// TIA Portal V17 export
// export: Created 2024-01-16T10:06:36.9177276Z, ExportSetting None, DisplayName Totally Integrated Automation Portal, DisplayVersion V17 Update 4, DisplayName TIA Portal Openness, DisplayVersion V17 Update 4, DisplayName TIA Portal Version Control Interface, DisplayVersion V17, DisplayName STEP 7 Professional, DisplayVersion V17 Update 4, DisplayName STEP 7 Safety, DisplayVersion V17, DisplayName WinCC Advanced / Unified PC, DisplayVersion V17 Update 4
FUNCTION "FC_FDIn" : Void   // FC13, F_LAD
// stored: AutoNumber false
BEGIN

REGION Network 1: GAS INLET VALVE OPEN
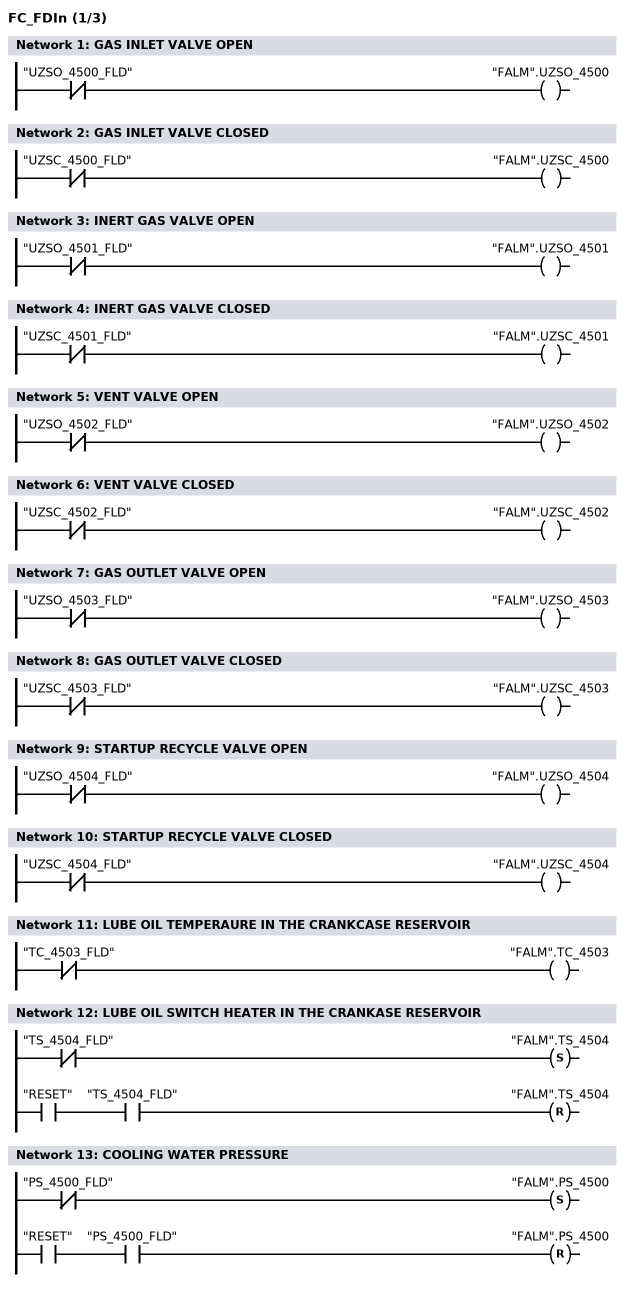
   RUNG wire#powerrail
      I_Contact( "UZSO_4500_FLD" )
      Coil( "FALM".UZSO_4500 )
   END_RUNG
   // the same network as SCL:
   "FALM".UZSO_4500 := NOT "UZSO_4500_FLD";
END_REGION

REGION Network 2: GAS INLET VALVE CLOSED
   RUNG wire#powerrail
      I_Contact( "UZSC_4500_FLD" )
      Coil( "FALM".UZSC_4500 )
   END_RUNG
   // the same network as SCL:
   "FALM".UZSC_4500 := NOT "UZSC_4500_FLD";
END_REGION

REGION Network 3: INERT GAS VALVE OPEN
   RUNG wire#powerrail
      I_Contact( "UZSO_4501_FLD" )
      Coil( "FALM".UZSO_4501 )
   END_RUNG
   // the same network as SCL:
   "FALM".UZSO_4501 := NOT "UZSO_4501_FLD";
END_REGION

REGION Network 4: INERT GAS VALVE CLOSED
   RUNG wire#powerrail
      I_Contact( "UZSC_4501_FLD" )
      Coil( "FALM".UZSC_4501 )
   END_RUNG
   // the same network as SCL:
   "FALM".UZSC_4501 := NOT "UZSC_4501_FLD";
END_REGION

REGION Network 5: VENT VALVE OPEN
   RUNG wire#powerrail
      I_Contact( "UZSO_4502_FLD" )
      Coil( "FALM".UZSO_4502 )
   END_RUNG
   // the same network as SCL:
   "FALM".UZSO_4502 := NOT "UZSO_4502_FLD";
END_REGION

REGION Network 6: VENT VALVE CLOSED
   RUNG wire#powerrail
      I_Contact( "UZSC_4502_FLD" )
      Coil( "FALM".UZSC_4502 )
   END_RUNG
   // the same network as SCL:
   "FALM".UZSC_4502 := NOT "UZSC_4502_FLD";
END_REGION

REGION Network 7: GAS OUTLET VALVE OPEN
   RUNG wire#powerrail
      I_Contact( "UZSO_4503_FLD" )
      Coil( "FALM".UZSO_4503 )
   END_RUNG
   // the same network as SCL:
   "FALM".UZSO_4503 := NOT "UZSO_4503_FLD";
END_REGION

REGION Network 8: GAS OUTLET VALVE CLOSED
   RUNG wire#powerrail
      I_Contact( "UZSC_4503_FLD" )
      Coil( "FALM".UZSC_4503 )
   END_RUNG
   // the same network as SCL:
   "FALM".UZSC_4503 := NOT "UZSC_4503_FLD";
END_REGION

REGION Network 9: STARTUP RECYCLE VALVE OPEN
   RUNG wire#powerrail
      I_Contact( "UZSO_4504_FLD" )
      Coil( "FALM".UZSO_4504 )
   END_RUNG
   // the same network as SCL:
   "FALM".UZSO_4504 := NOT "UZSO_4504_FLD";
END_REGION

REGION Network 10: STARTUP RECYCLE VALVE CLOSED
   RUNG wire#powerrail
      I_Contact( "UZSC_4504_FLD" )
      Coil( "FALM".UZSC_4504 )
   END_RUNG
   // the same network as SCL:
   "FALM".UZSC_4504 := NOT "UZSC_4504_FLD";
END_REGION

REGION Network 11: LUBE OIL TEMPERAURE IN THE CRANKCASE RESERVOIR
   RUNG wire#powerrail
      I_Contact( "TC_4503_FLD" )
      Coil( "FALM".TC_4503 )
   END_RUNG
   // the same network as SCL:
   "FALM".TC_4503 := NOT "TC_4503_FLD";
END_REGION

REGION Network 12: LUBE OIL SWITCH HEATER IN THE CRANKASE RESERVOIR
   RUNG wire#powerrail
      I_Contact( "TS_4504_FLD" )
      S_Coil( "FALM".TS_4504 )
   END_RUNG
   RUNG wire#powerrail
      Contact( "RESET" )
      Contact( "TS_4504_FLD" )
      R_Coil( "FALM".TS_4504 )
   END_RUNG
   // the same network as SCL:
   IF NOT "TS_4504_FLD" THEN "FALM".TS_4504 := TRUE; END_IF;
   IF "RESET" AND "TS_4504_FLD" THEN "FALM".TS_4504 := FALSE; END_IF;
END_REGION

REGION Network 13: COOLING WATER PRESSURE
   RUNG wire#powerrail
      I_Contact( "PS_4500_FLD" )
      S_Coil( "FALM".PS_4500 )
   END_RUNG
   RUNG wire#powerrail
      Contact( "RESET" )
      Contact( "PS_4500_FLD" )
      R_Coil( "FALM".PS_4500 )
   END_RUNG
   // the same network as SCL:
   IF NOT "PS_4500_FLD" THEN "FALM".PS_4500 := TRUE; END_IF;
   IF "RESET" AND "PS_4500_FLD" THEN "FALM".PS_4500 := FALSE; END_IF;
END_REGION

REGION Network 14: OUTLET GAS PRESSURE
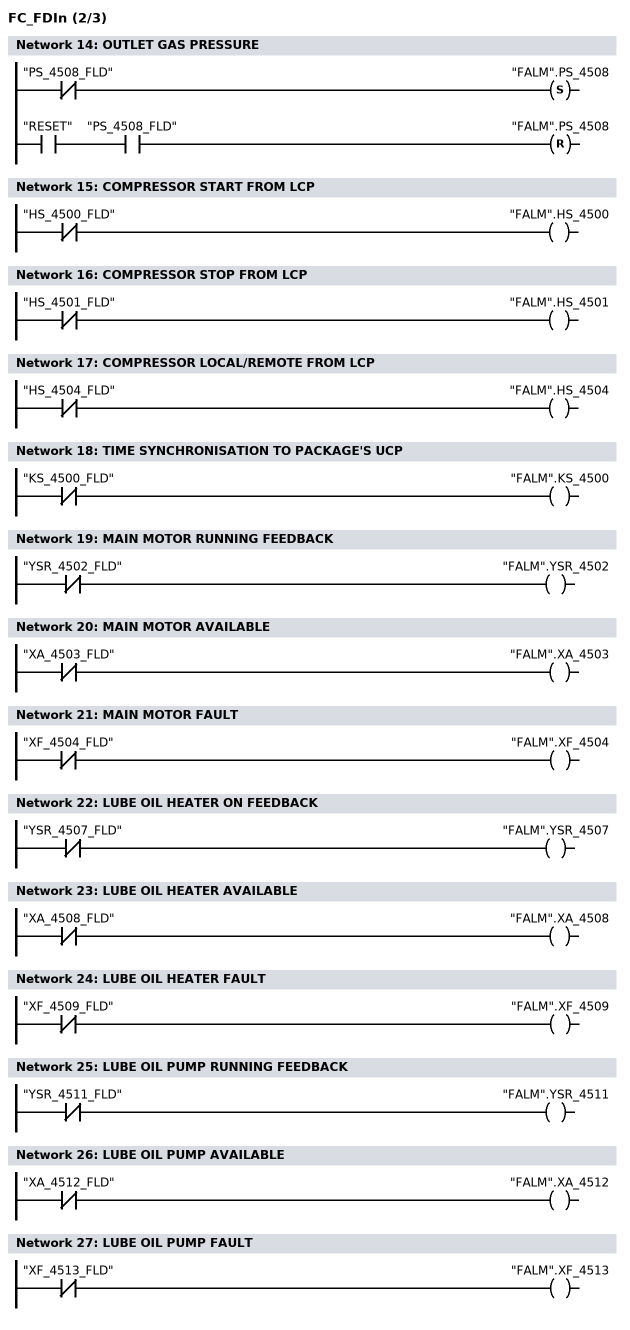
   RUNG wire#powerrail
      I_Contact( "PS_4508_FLD" )
      S_Coil( "FALM".PS_4508 )
   END_RUNG
   RUNG wire#powerrail
      Contact( "RESET" )
      Contact( "PS_4508_FLD" )
      R_Coil( "FALM".PS_4508 )
   END_RUNG
   // the same network as SCL:
   IF NOT "PS_4508_FLD" THEN "FALM".PS_4508 := TRUE; END_IF;
   IF "RESET" AND "PS_4508_FLD" THEN "FALM".PS_4508 := FALSE; END_IF;
END_REGION

REGION Network 15: COMPRESSOR START FROM LCP
   RUNG wire#powerrail
      I_Contact( "HS_4500_FLD" )
      Coil( "FALM".HS_4500 )
   END_RUNG
   // the same network as SCL:
   "FALM".HS_4500 := NOT "HS_4500_FLD";
END_REGION

REGION Network 16: COMPRESSOR STOP FROM LCP
   RUNG wire#powerrail
      I_Contact( "HS_4501_FLD" )
      Coil( "FALM".HS_4501 )
   END_RUNG
   // the same network as SCL:
   "FALM".HS_4501 := NOT "HS_4501_FLD";
END_REGION

REGION Network 17: COMPRESSOR LOCAL/REMOTE FROM LCP
   RUNG wire#powerrail
      I_Contact( "HS_4504_FLD" )
      Coil( "FALM".HS_4504 )
   END_RUNG
   // the same network as SCL:
   "FALM".HS_4504 := NOT "HS_4504_FLD";
END_REGION

REGION Network 18: TIME SYNCHRONISATION TO PACKAGE'S UCP
   RUNG wire#powerrail
      I_Contact( "KS_4500_FLD" )
      Coil( "FALM".KS_4500 )
   END_RUNG
   // the same network as SCL:
   "FALM".KS_4500 := NOT "KS_4500_FLD";
END_REGION

REGION Network 19: MAIN MOTOR RUNNING FEEDBACK
   RUNG wire#powerrail
      I_Contact( "YSR_4502_FLD" )
      Coil( "FALM".YSR_4502 )
   END_RUNG
   // the same network as SCL:
   "FALM".YSR_4502 := NOT "YSR_4502_FLD";
END_REGION

REGION Network 20: MAIN MOTOR AVAILABLE
   RUNG wire#powerrail
      I_Contact( "XA_4503_FLD" )
      Coil( "FALM".XA_4503 )
   END_RUNG
   // the same network as SCL:
   "FALM".XA_4503 := NOT "XA_4503_FLD";
END_REGION

REGION Network 21: MAIN MOTOR FAULT
   RUNG wire#powerrail
      I_Contact( "XF_4504_FLD" )
      Coil( "FALM".XF_4504 )
   END_RUNG
   // the same network as SCL:
   "FALM".XF_4504 := NOT "XF_4504_FLD";
END_REGION

REGION Network 22: LUBE OIL HEATER ON FEEDBACK
   RUNG wire#powerrail
      I_Contact( "YSR_4507_FLD" )
      Coil( "FALM".YSR_4507 )
   END_RUNG
   // the same network as SCL:
   "FALM".YSR_4507 := NOT "YSR_4507_FLD";
END_REGION

REGION Network 23: LUBE OIL HEATER AVAILABLE
   RUNG wire#powerrail
      I_Contact( "XA_4508_FLD" )
      Coil( "FALM".XA_4508 )
   END_RUNG
   // the same network as SCL:
   "FALM".XA_4508 := NOT "XA_4508_FLD";
END_REGION

REGION Network 24: LUBE OIL HEATER FAULT
   RUNG wire#powerrail
      I_Contact( "XF_4509_FLD" )
      Coil( "FALM".XF_4509 )
   END_RUNG
   // the same network as SCL:
   "FALM".XF_4509 := NOT "XF_4509_FLD";
END_REGION

REGION Network 25: LUBE OIL PUMP RUNNING FEEDBACK
   RUNG wire#powerrail
      I_Contact( "YSR_4511_FLD" )
      Coil( "FALM".YSR_4511 )
   END_RUNG
   // the same network as SCL:
   "FALM".YSR_4511 := NOT "YSR_4511_FLD";
END_REGION

REGION Network 26: LUBE OIL PUMP AVAILABLE
   RUNG wire#powerrail
      I_Contact( "XA_4512_FLD" )
      Coil( "FALM".XA_4512 )
   END_RUNG
   // the same network as SCL:
   "FALM".XA_4512 := NOT "XA_4512_FLD";
END_REGION

REGION Network 27: LUBE OIL PUMP FAULT
   RUNG wire#powerrail
      I_Contact( "XF_4513_FLD" )
      Coil( "FALM".XF_4513 )
   END_RUNG
   // the same network as SCL:
   "FALM".XF_4513 := NOT "XF_4513_FLD";
END_REGION

REGION Network 28: PLC CABINET - HIGH TEMPERATURE
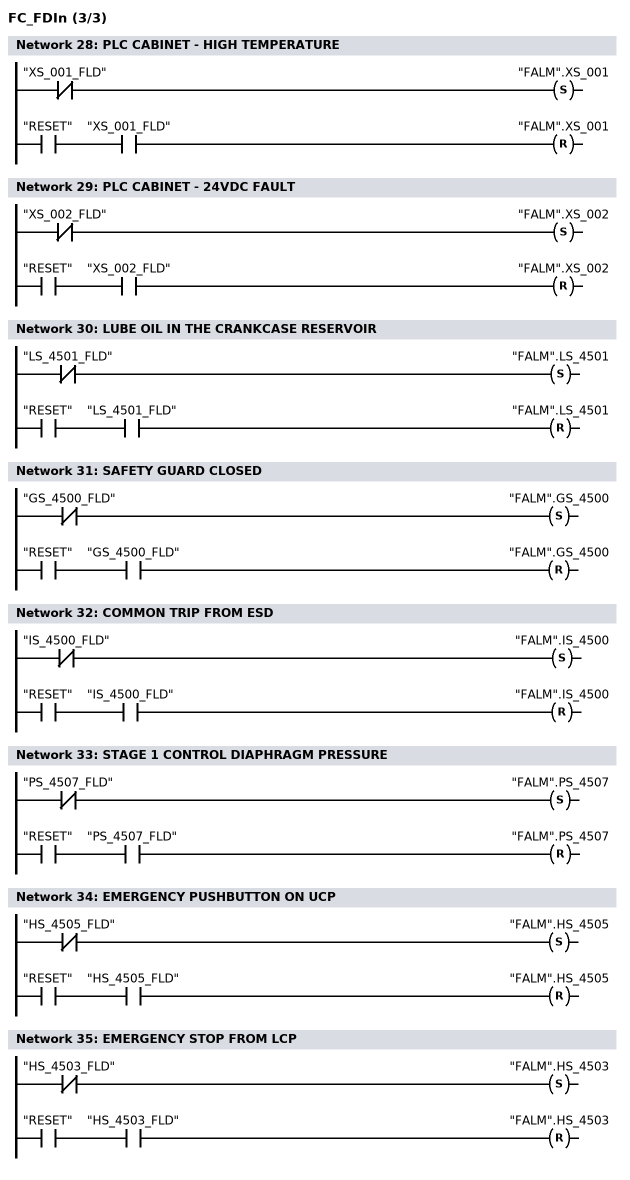
   RUNG wire#powerrail
      I_Contact( "XS_001_FLD" )
      S_Coil( "FALM".XS_001 )
   END_RUNG
   RUNG wire#powerrail
      Contact( "RESET" )
      Contact( "XS_001_FLD" )
      R_Coil( "FALM".XS_001 )
   END_RUNG
   // the same network as SCL:
   IF NOT "XS_001_FLD" THEN "FALM".XS_001 := TRUE; END_IF;
   IF "RESET" AND "XS_001_FLD" THEN "FALM".XS_001 := FALSE; END_IF;
END_REGION

REGION Network 29: PLC CABINET - 24VDC FAULT
   RUNG wire#powerrail
      I_Contact( "XS_002_FLD" )
      S_Coil( "FALM".XS_002 )
   END_RUNG
   RUNG wire#powerrail
      Contact( "RESET" )
      Contact( "XS_002_FLD" )
      R_Coil( "FALM".XS_002 )
   END_RUNG
   // the same network as SCL:
   IF NOT "XS_002_FLD" THEN "FALM".XS_002 := TRUE; END_IF;
   IF "RESET" AND "XS_002_FLD" THEN "FALM".XS_002 := FALSE; END_IF;
END_REGION

REGION Network 30: LUBE OIL IN THE CRANKCASE RESERVOIR
   RUNG wire#powerrail
      I_Contact( "LS_4501_FLD" )
      S_Coil( "FALM".LS_4501 )
   END_RUNG
   RUNG wire#powerrail
      Contact( "RESET" )
      Contact( "LS_4501_FLD" )
      R_Coil( "FALM".LS_4501 )
   END_RUNG
   // the same network as SCL:
   IF NOT "LS_4501_FLD" THEN "FALM".LS_4501 := TRUE; END_IF;
   IF "RESET" AND "LS_4501_FLD" THEN "FALM".LS_4501 := FALSE; END_IF;
END_REGION

REGION Network 31: SAFETY GUARD CLOSED
   RUNG wire#powerrail
      I_Contact( "GS_4500_FLD" )
      S_Coil( "FALM".GS_4500 )
   END_RUNG
   RUNG wire#powerrail
      Contact( "RESET" )
      Contact( "GS_4500_FLD" )
      R_Coil( "FALM".GS_4500 )
   END_RUNG
   // the same network as SCL:
   IF NOT "GS_4500_FLD" THEN "FALM".GS_4500 := TRUE; END_IF;
   IF "RESET" AND "GS_4500_FLD" THEN "FALM".GS_4500 := FALSE; END_IF;
END_REGION

REGION Network 32: COMMON TRIP FROM ESD
   RUNG wire#powerrail
      I_Contact( "IS_4500_FLD" )
      S_Coil( "FALM".IS_4500 )
   END_RUNG
   RUNG wire#powerrail
      Contact( "RESET" )
      Contact( "IS_4500_FLD" )
      R_Coil( "FALM".IS_4500 )
   END_RUNG
   // the same network as SCL:
   IF NOT "IS_4500_FLD" THEN "FALM".IS_4500 := TRUE; END_IF;
   IF "RESET" AND "IS_4500_FLD" THEN "FALM".IS_4500 := FALSE; END_IF;
END_REGION

REGION Network 33: STAGE 1 CONTROL DIAPHRAGM PRESSURE
   RUNG wire#powerrail
      I_Contact( "PS_4507_FLD" )
      S_Coil( "FALM".PS_4507 )
   END_RUNG
   RUNG wire#powerrail
      Contact( "RESET" )
      Contact( "PS_4507_FLD" )
      R_Coil( "FALM".PS_4507 )
   END_RUNG
   // the same network as SCL:
   IF NOT "PS_4507_FLD" THEN "FALM".PS_4507 := TRUE; END_IF;
   IF "RESET" AND "PS_4507_FLD" THEN "FALM".PS_4507 := FALSE; END_IF;
END_REGION

REGION Network 34: EMERGENCY PUSHBUTTON ON UCP
   RUNG wire#powerrail
      I_Contact( "HS_4505_FLD" )
      S_Coil( "FALM".HS_4505 )
   END_RUNG
   RUNG wire#powerrail
      Contact( "RESET" )
      Contact( "HS_4505_FLD" )
      R_Coil( "FALM".HS_4505 )
   END_RUNG
   // the same network as SCL:
   IF NOT "HS_4505_FLD" THEN "FALM".HS_4505 := TRUE; END_IF;
   IF "RESET" AND "HS_4505_FLD" THEN "FALM".HS_4505 := FALSE; END_IF;
END_REGION

REGION Network 35: EMERGENCY STOP FROM LCP
   RUNG wire#powerrail
      I_Contact( "HS_4503_FLD" )
      S_Coil( "FALM".HS_4503 )
   END_RUNG
   RUNG wire#powerrail
      Contact( "RESET" )
      Contact( "HS_4503_FLD" )
      R_Coil( "FALM".HS_4503 )
   END_RUNG
   // the same network as SCL:
   IF NOT "HS_4503_FLD" THEN "FALM".HS_4503 := TRUE; END_IF;
   IF "RESET" AND "HS_4503_FLD" THEN "FALM".HS_4503 := FALSE; END_IF;
END_REGION
END_FUNCTION
